{attribute 'qualified_only'}
{attribute 'strict'}
{attribute 'to_string'}
TYPE
ST180_Pnp_e :
(
    RESET := 0, // Reset

    INIT := 100, // Initialisieren 
    Init_HomeVertical_02,
    Init_Vertical_02_Up,
    Init_HomeVertical_10,
    Init_Vertical_10_Down,
    Init_HomeHorizontal,
    Init_HorizontalToTrack,
    Init_check_if_pces_handled,

    READY := 999,  // READY to Start, Init Done 
    START := 1000, // Start Zyklisch

    waitOnMover,     // wait until the mover is there
    MOVER_NEEDED_OP, // Ab here, a mover in position is needed to perform the action

    lift_piece_and_down_to_pick,        // lift the piece with 180.10Z and go down simultaneously with 180.02Z
    close_griper_pick_piece,            // close the griper to pick the piece
    clamp_down_maintain_piece,          // the clamp (niederhalter) goes down and hold the piece in place
    take_out_piece_and_put_down_lifter, // 180.02Z goes up with the piece, 180.10Z goes down

    SYNC_MOVER_LEAVE, // MoverMan need to take the mover
    MOVER_FREE_OP,    // here, operation without mover can be done.

    hor_move_to_extraction_pipe, // 180.01Y move to the extraction pipe
    ver_down_in_pipe,            // 180.02Z move down to a secure position to release the piece
    open_griper_put_piece,
    clamp_up_to_rest_position,
    ver_up_empty,					// 180.02z goes up without piece
    hor_to_track_pos,

    DONE := 8000,  // Ablauf beendet 
    ERROR := 9000, // Fehler 
    _max
);
END_TYPE

(*
back to shuttle
check level NIO Box
*)

(* stored: Version 1.1.0.1, ProductVersion 3.1.4024.6
   EnumerationTextList ST180_Pnp_e: Id {d7db67ab-cc04-42aa-8dc6-05b0e0594efd} *)
